// TwinCAT 3 PLC project lclsPLCMotionTest
// ProgramVersion: 3.1.4026.17
// libraries:
//   LCLS General, * (SLAC)
//   LCLS_OOPMotion, * (SLAC)
//   Tc2_MC2, * (Beckhoff Automation GmbH)
//   Tc2_NC, * (Beckhoff Automation GmbH)
//   Tc2_Standard, * (Beckhoff Automation GmbH)
//   Tc2_System, * (Beckhoff Automation GmbH)
// project tree:
//   DUTs/ ENUM_AxisStates.TcDUT (not stored)
//   GVLs/ GVL_Axes.TcGVL
//   / PlcTask.TcTTO (not stored)
//   POUs/ MAIN.TcPOU
// real-time tasks:
//   TASK PlcTask: cycle T#10ms, priority 20, ADS port 350
// motion (NC):
//   TASK NC-Task 1 SAF: cycle T#2ms, priority 4, ADS port 501
//   TASK NC-Task 1 SVB: cycle T#10ms, priority 8, ADS port 511
//   AXIS Axis 1 (id 1)
//   AXIS Axis 2 (id 2)
//   AXIS Axis 3 (id 3)
//   AXIS Axis 4 (id 4)
// variable links:
//   (this object) <-> NC-Task 1 SAF/Axes/Axis 1
//     PlcTask Inputs/GVL_Axes.Axes[1].NcToPlc <-> Outputs/ToPlc
//     PlcTask Outputs/GVL_Axes.Axes[1].PlcToNc <-> Inputs/FromPlc
//   (this object) <-> NC-Task 1 SAF/Axes/Axis 2
//     PlcTask Inputs/GVL_Axes.Axes[2].NcToPlc <-> Outputs/ToPlc
//     PlcTask Outputs/GVL_Axes.Axes[2].PlcToNc <-> Inputs/FromPlc
//   (this object) <-> NC-Task 1 SAF/Axes/Axis 3
//     PlcTask Inputs/GVL_Axes.Axes[3].NcToPlc <-> Outputs/ToPlc
//     PlcTask Outputs/GVL_Axes.Axes[3].PlcToNc <-> Inputs/FromPlc
//   (this object) <-> NC-Task 1 SAF/Axes/Axis 4
//     PlcTask Inputs/GVL_Axes.Axes[4].NcToPlc <-> Outputs/ToPlc
//     PlcTask Outputs/GVL_Axes.Axes[4].PlcToNc <-> Inputs/FromPlc

// ---- GVLs/GVL_Axes.TcGVL
{attribute 'qualified_only'}
VAR_GLOBAL
    Axes :  ARRAY[1..2] OF AXIS_REF;
END_VAR

// ---- POUs/MAIN.TcPOU
PROGRAM MAIN
VAR
    fbPersistentDataStorage : FB_PersistentDataStorage;
	{attribute 'pytmc' := '
		axis-link: GVL_Axes.Axes[1]
		pv: TST:MOTION:SLITX
	'}
   	slitX : FB_MotionStageNC(	sName := 'slitX',
                                        AxisRef := GVL_Axes.Axes[1],
                                        iPersistentDataStorage := fbPersistentDataStorage
                                    ) ;
	{attribute 'pytmc' := '
		axis-link: GVL_Axes.Axes[2]
		pv: TST:MOTION:SLITY
	'}
   	slitY : FB_MotionStageNC(	sName := 'slitY',
                                        AxisRef := GVL_Axes.Axes[2],
                                        iPersistentDataStorage := fbPersistentDataStorage
                                    ) ;
	{attribute 'pytmc' := '
		axis-link: GVL_Axes.Axes[3]
		pv: TST:MOTION:SLITZ
	'}
   	slitZ : FB_MotionStageNC(	sName := 'slitZ',
                                        AxisRef := GVL_Axes.Axes[3],
                                        iPersistentDataStorage := fbPersistentDataStorage
                                    ) ;
   	dummy : FB_MotionStageNC(	sName := 'dummy',
                                        AxisRef := GVL_Axes.Axes[4],
                                        iPersistentDataStorage := fbPersistentDataStorage
                                    ) ;
END_VAR

fbPersistentDataStorage();
slitX();
slitY();
slitZ();
dummy();

END_PROGRAM
